(*
Nazwa:			E_CapFeederState
Opis:			Stany sortera nasadek
Wersja:			v0.1
Data:			2018-10-10
Autor:			DP
Urzadzenia:		
Konfiguracja:	
Info:
*)


TYPE E_WickFeederSorterState :
(
	eDisabled:=0,  		//Wyłączona
	eError:=1,			//Błąd
	eManualMovement:=2, //Tryb serwisowy
	eHoming:=3,			//Bazowanie
	eHomingDone:=4, 	//Koniec bazowania
	eReady:=5,			//Gotowość
	eSleeveLowLevel:=6, //Praca, Niski poziom
	eSorting:=7,		//Praca
	eSleeveFull:=8,		//Zapełniona
	ePreparingToDisable:=10 (*NOWY*) //Przygotowanie do wyłączenia
):=eDisabled;
END_TYPE

(* stored: Version 1.2.0.0, ProductVersion 3.1.4026.13, FileIdentifier 8b2f994d96752568194cbeec1310d4c9ba6615a0, FileSignature 5f1288466632272d56e32c2edea82f3eea38fa630e5686025fc97a957bb5f48c45d658f521bea3738f318012977fedef1f59f555fb44a071d4190414e1348d7f3d3c19a1b9cab3aa9981be06fdc7708276740017d78b690bcaf042fadf8c2e7805e75f55da94ed47eab5bcba891d113b190f4cc83ade5e3244df361f839c04388ba82278a29ab127cc2682a5682e00072f46411cb600f3eede454cbd71cf8eef3a9e46229a3381f081bd2d2748b3c9526964cdefc278fb4c6f9e51c3151eb6ad1899d591a186adbf8683e20b86e5818449baf6efb56ed75ab525e531ca8c070ff12716820baa290bba6991277f4cedd9d320a6fc6ef7d2030cba10916d40eee0
   DUT E_WickFeederSorterState: Id {365176ae-91f2-47f6-aee4-492c92097a54} *)
